{attribute 'linkalways'} 
{attribute 'no_explicit_call' := 'This FB is a CLASS and must be accessed using methods or properties'}
{attribute 'enable_dynamic_creation'}
FUNCTION_BLOCK _LWORD EXTENDS IntegerDatatypeBase
VAR
	localData : LWORD;
	activeData : REFERENCE TO LWORD REF= localData;
END_VAR

PROPERTY PUBLIC Address : PVOID
GET
Address := ADR(activeData);
END_GET
END_PROPERTY

METHOD PUBLIC ClearReference
VAR_INPUT
END_VAR
activeData REF= localData;
END_METHOD

METHOD PUBLIC Clone : I_Datatype
VAR
    pClone : POINTER TO _LWORD;
END_VAR
pClone := __NEW(_LWORD(InitialValue := Value));
Clone := pClone^;
END_METHOD

PROPERTY PUBLIC Datatype : T_MAXSTRING
GET
Datatype := 'LWORD';
END_GET
END_PROPERTY

METHOD FB_init : BOOL
VAR_INPUT
	bInitRetains : BOOL; // if TRUE, the retain variables are initialized (warm start / cold start)
	bInCopyCode : BOOL;  // if TRUE, the instance afterwards gets moved WORDo the copy code (online change)
	InitialValue : LWORD;
END_VAR
localData := InitialValue;
END_METHOD

PROPERTY PUBLIC IsSigned : BOOL
GET
IsSigned := FALSE;
END_GET
END_PROPERTY

PROPERTY PUBLIC LowerBound : LWORD
GET
LowerBound := DatatypeLimits.LWORD_LOWER_LIMIT;
END_GET
END_PROPERTY

METHOD PUBLIC MakeReferenceTo
VAR_INPUT
	ReferenceTarget : REFERENCE TO LWORD;
END_VAR
activeData REF= ReferenceTarget;
END_METHOD

METHOD PROTECTED SerializeLowerbound
VAR_INPUT
	Serializer : I_Serializer;
END_VAR
Serializer.AddLword(Lowerbound);
END_METHOD

METHOD PROTECTED SerializeUpperbound
VAR_INPUT
	Serializer : I_Serializer;
END_VAR
Serializer.AddLword(Upperbound);
END_METHOD

METHOD PUBLIC SerializeWith
VAR_INPUT
	Serializer : I_Serializer;
END_VAR
Serializer.AddLword(activeData);
END_METHOD

PROPERTY PUBLIC Size : UDINT
GET
Size := SIZEOF(activeData);
END_GET
END_PROPERTY

METHOD TryDeserializeFrom : BOOL
VAR_INPUT
	Deserializer : I_Deserializer;
	Feedback : I_DeserializerFeedback;
END_VAR
TryDeserializeFrom := Deserializer.TryGetLword(activeData, Feedback);
END_METHOD

METHOD TryMakeReferenceTo : BOOL
VAR_INPUT
	Target : I_Datatype;
END_VAR
VAR
	pTargetData : POINTER TO LWORD;
END_VAR
IF NOT (Target.Datatype = Datatype) THEN
	RETURN;
END_IF

pTargetData := Target.Address;
activeData REF= pTargetData^;
TryMakeReferenceTo := TRUE;
END_METHOD

PROPERTY PUBLIC UpperBound : LWORD
GET
UpperBound :=  DatatypeLimits.LWORD_UPPER_LIMIT;
END_GET
END_PROPERTY

PROPERTY PUBLIC Value : LWORD
GET
Value := activeData;
END_GET
SET
activeData := Value;
END_SET
END_PROPERTY

END_FUNCTION_BLOCK

(* stored: Version 1.1.0.1, ProductVersion 3.1.4024.12
   POU _LWORD: Id {83eb2057-61c3-0f5c-2bbd-2c1a0c4bcdbb}, SpecialFunc None
   Folder Constructor: Id {76a599ac-f355-0c91-3411-2c4573633eb2}
   Folder Protected: Id {944a4539-c918-0a7b-2b1f-c61cad3b8df0}
   Property Address: Id {3ea38e9d-e5b4-08f8-3bac-d50de01d8088}
   Get Get: Id {4c3c2f62-1325-05ee-2e66-2b5f5411ac84}
   Method ClearReference: Id {10b74754-dd3d-0784-2dc0-bc9aaaa6dff2}
   Method Clone: Id {70ec616f-2c61-064a-2209-68affc8cda70}
   Property Datatype: Id {f1ea044d-8243-0a57-0c7e-1f8798251cf8}
   Get Get: Id {7c6d7a65-de1e-06bb-2224-776a3f729bc6}
   Method FB_init: Id {6fbd1526-f642-03c9-1957-3df80912e78f}
   Property IsSigned: Id {2a485424-884d-0894-2c06-375b2616271e}
   Get Get: Id {cbc87458-11d1-0a1b-173b-3d185c3cd538}
   Property LowerBound: Id {c4400076-e1a9-0cf7-2ba2-1351544eec14}
   Get Get: Id {be29f02c-45c3-07fa-2210-b1cf141d0854}
   Method MakeReferenceTo: Id {22dc0f3b-b797-03c0-006f-7c61fb3682bc}
   Method SerializeLowerbound: Id {a582afe9-1aaf-0ab1-2c9a-35d9e67f192f}
   Method SerializeUpperbound: Id {5f4c0310-6d98-0d57-2a8a-5fb9a16cecec}
   Method SerializeWith: Id {43957286-f88e-05ee-30ce-fc0a753ce5f1}
   Property Size: Id {e6a57ecf-e117-0957-19ab-e82010e77df9}
   Get Get: Id {e9dcdc74-ac46-04bd-0982-1d0e341f3ca2}
   Method TryDeserializeFrom: Id {0e99a354-8f0e-0ad8-03af-ecb45be70e2a}
   Method TryMakeReferenceTo: Id {7534ac8b-b439-087c-0eca-0e1f7561613f}
   Property UpperBound: Id {8960f733-ee11-0800-1b8e-413b576219a5}
   Get Get: Id {810e74c1-1278-03b7-144f-3628788e50dc}
   Property Value: Id {32408784-0d34-0b64-3e25-e04ead8e7528}
   Get Get: Id {4b97d08e-c899-0a71-3b3b-f66d8e13a09d}
   Set Set: Id {4a2d1657-4af8-0535-24f3-4c03181dcf25} *)
